LIN {X 0,Y 97.337,Z 845.58,A -85,B 0,C 180,E1 -28950.042,E2 -28950.042} C_VEL
LIN {X 0,Y 109.407,Z 841.998,A -85,B 0,C 180,E1 -28954.063,E2 -28954.063} C_VEL
LIN {X 0,Y 115.747,Z 839.589,A -85,B 0,C 180,E1 -28955.608,E2 -28955.608} C_VEL
LIN {X 0,Y 117.858,Z 838.675,A -85,B 0,C 180,E1 -28956.642,E2 -28956.642} C_VEL
LIN {X 0,Y 108.454,Z 842.054,A -85,B 0,C 180,E1 -28959.119,E2 -28959.119} C_VEL
LIN {X 0,Y 95.133,Z 845.441,A -85,B 0,C 180,E1 -28963.809,E2 -28963.809} C_VEL
LIN {X 0,Y 86.195,Z 846.778,A -85,B 0,C 180,E1 -28968.064,E2 -28968.064} C_VEL
LIN {X 0,Y 76.127,Z 847.276,A -85,B 0,C 180,E1 -28974.702,E2 -28974.702} C_VEL
LIN {X 0,Y 70.276,Z 846.865,A -85,B 0,C 180,E1 -28980.071,E2 -28980.071} C_VEL
LIN {X 0,Y 63.905,Z 845.572,A -85,B 0,C 180,E1 -28988.222,E2 -28988.222} C_VEL
LIN {X 0,Y 57.877,Z 842.432,A -85,B 0,C 180,E1 -29001.363,E2 -29001.363} C_VEL
LIN {X 0,Y 55.288,Z 838.085,A -85,B 0,C 180,E1 -29014.89,E2 -29014.89} C_VEL
LIN {X 0,Y 55.324,Z 833.064,A -85,B 0,C 180,E1 -29026.92,E2 -29026.92} C_VEL
LIN {X 0,Y 56.871,Z 827.685,A -85,B 0,C 180,E1 -29036.869,E2 -29036.869} C_VEL
LIN {X 0,Y 59.908,Z 820.393,A -85,B 0,C 180,E1 -29047.051,E2 -29047.051} C_VEL
LIN {X 0,Y 60.928,Z 818.162,A -85,B 0,C 180,E1 -29049.601,E2 -29049.601} C_VEL
LIN {X 0,Y 62.142,Z 814.385,A -85,B 0,C 180,E1 -29053.604,E2 -29053.604} C_VEL
LIN {X 0,Y 62.854,Z 807.647,A -85,B 0,C 180,E1 -29060.19,E2 -29060.19} C_VEL
LIN {X 0,Y 64.057,Z 800.304,A -85,B 0,C 180,E1 -29066.256,E2 -29066.256} C_VEL
LIN {X 0,Y 65.919,Z 795.617,A -85,B 0,C 180,E1 -29069.117,E2 -29069.117} C_VEL
LIN {X 0,Y 70.749,Z 785.494,A -85,B 0,C 180,E1 -29073.493,E2 -29073.493} C_VEL
LIN {X 0,Y 71.926,Z 778.933,A -85,B 0,C 180,E1 -29076.609,E2 -29076.609} C_VEL
LIN {X 0,Y 70.875,Z 778.62,A -85,B 0,C 180,E1 -29077.433,E2 -29077.433} C_VEL
LIN {X 0,Y 64.084,Z 778.084,A -85,B 0,C 180,E1 -29082.673,E2 -29082.673} C_VEL
LIN {X 0,Y 59.157,Z 776.717,A -85,B 0,C 180,E1 -29088.122,E2 -29088.122} C_VEL
LIN {X 0,Y 54.146,Z 776.16,A -85,B 0,C 180,E1 -29094.693,E2 -29094.693} C_VEL
LIN {X 0,Y 52.689,Z 774.473,A -85,B 0,C 180,E1 -29098.644,E2 -29098.644} C_VEL
LIN {X 0,Y 52.676,Z 779.282,A -85,B 0,C 180,E1 -29111.848,E2 -29111.848} C_VEL
LIN {X 0,Y 55.548,Z 783.057,A -85,B 0,C 180,E1 -29125.331,E2 -29125.331} C_VEL
LIN {X 0,Y 61,Z 785.546,A -85,B 0,C 180,E1 -29137.185,E2 -29137.185} C_VEL
LIN {X 0,Y 65.827,Z 786.444,A -85,B 0,C 180,E1 -29143.932,E2 -29143.932} C_VEL
LIN {X 0,Y 71.43,Z 786.807,A -85,B 0,C 180,E1 -29149.721,E2 -29149.721} C_VEL
LIN {X 0,Y 77.758,Z 786.531,A -85,B 0,C 180,E1 -29154.815,E2 -29154.815} C_VEL
LIN {X 0,Y 86.181,Z 785.381,A -85,B 0,C 180,E1 -29160.001,E2 -29160.001} C_VEL
LIN {X 0,Y 95.086,Z 783.29,A -85,B 0,C 180,E1 -29164.239,E2 -29164.239} C_VEL
LIN {X 0,Y 98.897,Z 782.143,A -85,B 0,C 180,E1 -29165.777,E2 -29165.777} C_VEL
LIN {X 0,Y 102.271,Z 781.127,A -85,B 0,C 180,E1 -29167.9,E2 -29167.9} C_VEL
LIN {X 0,Y 103.122,Z 781.36,A -85,B 0,C 180,E1 -29171.798,E2 -29171.798} C_VEL
LIN {X 0,Y 102.209,Z 782.608,A -85,B 0,C 180,E1 -29175.965,E2 -29175.965} C_VEL
LIN {X 0,Y 100.508,Z 784.208,A -85,B 0,C 180,E1 -29179.374,E2 -29179.374} C_VEL
LIN {X 0,Y 91.817,Z 788.201,A -85,B 0,C 180,E1 -29183.284,E2 -29183.284} C_VEL
LIN {X 0,Y 80.528,Z 792.377,A -85,B 0,C 180,E1 -29189.217,E2 -29189.217} C_VEL
LIN {X 0,Y 70.349,Z 795.196,A -85,B 0,C 180,E1 -29196.94,E2 -29196.94} C_VEL
LIN {X 0,Y 66.904,Z 796.068,A -85,B 0,C 180,E1 -29200.409,E2 -29200.409} C_VEL
LIN {X 0,Y 61.403,Z 806.889,A -85,B 0,C 180,E1 -29206.623,E2 -29206.623} C_VEL
LIN {X 0,Y 56.665,Z 815.69,A -85,B 0,C 180,E1 -29213.901,E2 -29213.901} C_VEL
LIN {X 0,Y 52.334,Z 824.279,A -85,B 0,C 180,E1 -29224.118,E2 -29224.118} C_VEL
LIN {X 0,Y 49.821,Z 831.224,A -85,B 0,C 180,E1 -29235.704,E2 -29235.704} C_VEL
LIN {X 0,Y 49.137,Z 835.892,A -85,B 0,C 180,E1 -29245.895,E2 -29245.895} C_VEL
LIN {X 0,Y 49.267,Z 838.605,A -85,B 0,C 180,E1 -29253.059,E2 -29253.059} C_VEL
LIN {X 0,Y 50.036,Z 842.482,A -85,B 0,C 180,E1 -29266.31,E2 -29266.31} C_VEL
LIN {X 0,Y 54.162,Z 845.868,A -85,B 0,C 180,E1 -29281.263,E2 -29281.263} C_VEL
LIN {X 0,Y 61.486,Z 847.824,A -85,B 0,C 180,E1 -29293.295,E2 -29293.295} C_VEL
LIN {X 0,Y 71.066,Z 848.501,A -85,B 0,C 180,E1 -29302.288,E2 -29302.288} C_VEL
LIN {X 0,Y 82.054,Z 847.895,A -85,B 0,C 180,E1 -29308.921,E2 -29308.921} C_VEL
LIN {X 0,Y 94,Z 845.97,A -85,B 0,C 180,E1 -29313.785,E2 -29313.785} C_VEL
LIN {X 0,Y 100.238,Z 844.484,A -85,B 0,C 180,E1 -29315.704,E2 -29315.704} C_VEL
LIN {X 0,Y 100.894,Z 844.252,A -85,B 0,C 180,E1 -29316.994,E2 -29316.994} C_VEL
LIN {X 0,Y 88.164,Z 846.641,A -85,B 0,C 180,E1 -29321.405,E2 -29321.405} C_VEL
LIN {X 0,Y 79.941,Z 847.375,A -85,B 0,C 180,E1 -29325.242,E2 -29325.242} C_VEL
LIN {X 0,Y 71.204,Z 847.416,A -85,B 0,C 180,E1 -29330.737,E2 -29330.737} C_VEL
LIN {X 0,Y 61.361,Z 846.218,A -85,B 0,C 180,E1 -29339.999,E2 -29339.999} C_VEL
LIN {X 0,Y 54.212,Z 843.827,A -85,B 0,C 180,E1 -29351.212,E2 -29351.212} C_VEL
LIN {X 0,Y 49.577,Z 840.062,A -85,B 0,C 180,E1 -29365.167,E2 -29365.167} C_VEL
LIN {X 0,Y 48.011,Z 835.37,A -85,B 0,C 180,E1 -29379.356,E2 -29379.356} C_VEL
LIN {X 0,Y 49.024,Z 829.528,A -85,B 0,C 180,E1 -29393.16,E2 -29393.16} C_VEL
LIN {X 0,Y 51.417,Z 823.332,A -85,B 0,C 180,E1 -29404.099,E2 -29404.099} C_VEL
LIN {X 0,Y 55.431,Z 815.299,A -85,B 0,C 180,E1 -29414.374,E2 -29414.374} C_VEL
LIN {X 0,Y 60.999,Z 805.035,A -85,B 0,C 180,E1 -29423.388,E2 -29423.388} C_VEL
LIN {X 0,Y 65.919,Z 795.617,A -85,B 0,C 180,E1 -29429.117,E2 -29429.117} C_VEL
LIN {X 0,Y 66.46,Z 793.686,A -85,B 0,C 180,E1 -29430.333,E2 -29430.333} C_VEL
LIN {X 0,Y 65.983,Z 790.673,A -85,B 0,C 180,E1 -29432.816,E2 -29432.816} C_VEL
LIN {X 0,Y 64.886,Z 786.315,A -85,B 0,C 180,E1 -29436.529,E2 -29436.529} C_VEL
LIN {X 0,Y 64.896,Z 785.615,A -85,B 0,C 180,E1 -29436.997,E2 -29436.997} C_VEL
LIN {X 0,Y 64.976,Z 784.515,A -85,B 0,C 180,E1 -29437.69,E2 -29437.69} C_VEL
LIN {X 0,Y 52.577,Z 782.682,A -85,B 0,C 180,E1 -29450.664,E2 -29450.664} C_VEL
LIN {X 0,Y 50.05,Z 781.938,A -85,B 0,C 180,E1 -29454.919,E2 -29454.919} C_VEL
LIN {X 0,Y 48.232,Z 780.916,A -85,B 0,C 180,E1 -29459.042,E2 -29459.042} C_VEL
LIN {X 0,Y 46.361,Z 780.459,A -85,B 0,C 180,E1 -29463.383,E2 -29463.383} C_VEL
LIN {X 0,Y 45.36,Z 778.621,A -85,B 0,C 180,E1 -29468.939,E2 -29468.939} C_VEL
LIN {X 0,Y 47.662,Z 782.726,A -85,B 0,C 180,E1 -29483.857,E2 -29483.857} C_VEL
LIN {X 0,Y 53.163,Z 785.8,A -85,B 0,C 180,E1 -29497.736,E2 -29497.736} C_VEL
LIN {X 0,Y 58.848,Z 787.189,A -85,B 0,C 180,E1 -29506.182,E2 -29506.182} C_VEL
LIN {X 0,Y 66.591,Z 787.888,A -85,B 0,C 180,E1 -29513.943,E2 -29513.943} C_VEL
LIN {X 0,Y 77.331,Z 787.449,A -85,B 0,C 180,E1 -29521.316,E2 -29521.316} C_VEL
LIN {X 0,Y 84.667,Z 786.379,A -85,B 0,C 180,E1 -29525.043,E2 -29525.043} C_VEL
LIN {X 0,Y 93.622,Z 784.354,A -85,B 0,C 180,E1 -29528.635,E2 -29528.635} C_VEL
LIN {X 0,Y 96.122,Z 783.845,A -85,B 0,C 180,E1 -29530.533,E2 -29530.533} C_VEL
LIN {X 0,Y 96.146,Z 784.213,A -85,B 0,C 180,E1 -29532.668,E2 -29532.668} C_VEL
LIN {X 0,Y 95.065,Z 785.304,A -85,B 0,C 180,E1 -29536.033,E2 -29536.033} C_VEL
LIN {X 0,Y 92.068,Z 786.659,A -85,B 0,C 180,E1 -29537.779,E2 -29537.779} C_VEL
LIN {X 0,Y 83.149,Z 789.928,A -85,B 0,C 180,E1 -29541.597,E2 -29541.597} C_VEL
LIN {X 0,Y 71.606,Z 793.148,A -85,B 0,C 180,E1 -29547.947,E2 -29547.947} C_VEL
LIN {X 0,Y 61.147,Z 795.333,A -85,B 0,C 180,E1 -29556.773,E2 -29556.773} C_VEL
LIN {X 0,Y 55.344,Z 805.988,A -85,B 0,C 180,E1 -29563.094,E2 -29563.094} C_VEL
LIN {X 0,Y 50.173,Z 814.923,A -85,B 0,C 180,E1 -29570.919,E2 -29570.919} C_VEL
LIN {X 0,Y 45.436,Z 823.576,A -85,B 0,C 180,E1 -29582.347,E2 -29582.347} C_VEL
LIN {X 0,Y 42.75,Z 830.558,A -85,B 0,C 180,E1 -29595.719,E2 -29595.719} C_VEL
LIN {X 0,Y 42.189,Z 836.105,A -85,B 0,C 180,E1 -29609.995,E2 -29609.995} C_VEL
LIN {X 0,Y 42.383,Z 839.021,A -85,B 0,C 180,E1 -29619.54,E2 -29619.54} C_VEL
LIN {X 0,Y 43.338,Z 841.409,A -85,B 0,C 180,E1 -29628.92,E2 -29628.92} C_VEL
LIN {X 0,Y 48.259,Z 845.009,A -85,B 0,C 180,E1 -29645.623,E2 -29645.623} C_VEL
LIN {X 0,Y 56.537,Z 847.275,A -85,B 0,C 180,E1 -29658.226,E2 -29658.226} C_VEL
LIN {X 0,Y 66.96,Z 848.237,A -85,B 0,C 180,E1 -29667.099,E2 -29667.099} C_VEL
LIN {X 0,Y 79.607,Z 847.804,A -85,B 0,C 180,E1 -29673.805,E2 -29673.805} C_VEL
LIN {X 0,Y 84.784,Z 847.24,A -85,B 0,C 180,E1 -29675.752,E2 -29675.752} C_VEL
LIN {X 0,Y 85.312,Z 847.12,A -85,B 0,C 180,E1 -29677.097,E2 -29677.097} C_VEL
LIN {X 0,Y 72,Z 847.759,A -85,B 0,C 180,E1 -29682.971,E2 -29682.971} C_VEL
LIN {X 0,Y 64.772,Z 847.344,A -85,B 0,C 180,E1 -29687.546,E2 -29687.546} C_VEL
LIN {X 0,Y 56.435,Z 846.07,A -85,B 0,C 180,E1 -29694.992,E2 -29694.992} C_VEL
LIN {X 0,Y 47.475,Z 842.995,A -85,B 0,C 180,E1 -29708.512,E2 -29708.512} C_VEL
LIN {X 0,Y 42.448,Z 838.838,A -85,B 0,C 180,E1 -29724.45,E2 -29724.45} C_VEL
LIN {X 0,Y 40.969,Z 834.012,A -85,B 0,C 180,E1 -29740.189,E2 -29740.189} C_VEL
LIN {X 0,Y 42.328,Z 827.781,A -85,B 0,C 180,E1 -29756.114,E2 -29756.114} C_VEL
LIN {X 0,Y 46.034,Z 819.842,A -85,B 0,C 180,E1 -29770.545,E2 -29770.545} C_VEL
LIN {X 0,Y 50.792,Z 811.433,A -85,B 0,C 180,E1 -29780.859,E2 -29780.859} C_VEL
LIN {X 0,Y 56.667,Z 801.359,A -85,B 0,C 180,E1 -29789.122,E2 -29789.122} C_VEL
LIN {X 0,Y 62.557,Z 790.472,A -85,B 0,C 180,E1 -29795,E2 -29795} C_VEL
LIN {X 0,Y 64.896,Z 785.615,A -85,B 0,C 180,E1 -29796.997,E2 -29796.997} C_VEL
LIN {X 0,Y 64.321,Z 784.532,A -85,B 0,C 180,E1 -29798.144,E2 -29798.144} C_VEL
LIN {X 0,Y 62.594,Z 784.124,A -85,B 0,C 180,E1 -29799.71,E2 -29799.71} C_VEL
LIN {X 0,Y 59.438,Z 784.737,A -85,B 0,C 180,E1 -29801.741,E2 -29801.741} C_VEL
LIN {X 0,Y 51.676,Z 787.896,A -85,B 0,C 180,E1 -29806.496,E2 -29806.496} C_VEL
LIN {X 0,Y 48.765,Z 788.348,A -85,B 0,C 180,E1 -29809.575,E2 -29809.575} C_VEL
LIN {X 0,Y 48.234,Z 788.279,A -85,B 0,C 180,E1 -29810.273,E2 -29810.273} C_VEL
LIN {X 0,Y 46.147,Z 787.8,A -85,B 0,C 180,E1 -29813.971,E2 -29813.971} C_VEL
LIN {X 0,Y 44.339,Z 786.87,A -85,B 0,C 180,E1 -29818.398,E2 -29818.398} C_VEL
LIN {X 0,Y 42.292,Z 786.267,A -85,B 0,C 180,E1 -29823.813,E2 -29823.813} C_VEL
LIN {X 0,Y 39.709,Z 783.567,A -85,B 0,C 180,E1 -29838.969,E2 -29838.969} C_VEL
LIN {X 0,Y 39.996,Z 782.339,A -85,B 0,C 180,E1 -29842.772,E2 -29842.772} C_VEL
LIN {X 0,Y 45.317,Z 785.818,A -85,B 0,C 180,E1 -29858.526,E2 -29858.526} C_VEL
LIN {X 0,Y 50.472,Z 787.442,A -85,B 0,C 180,E1 -29867.104,E2 -29867.104} C_VEL
LIN {X 0,Y 56.536,Z 788.528,A -85,B 0,C 180,E1 -29874.011,E2 -29874.011} C_VEL
LIN {X 0,Y 63.833,Z 789.022,A -85,B 0,C 180,E1 -29880.001,E2 -29880.001} C_VEL
LIN {X 0,Y 73.049,Z 788.763,A -85,B 0,C 180,E1 -29885.522,E2 -29885.522} C_VEL
LIN {X 0,Y 85.904,Z 787.008,A -85,B 0,C 180,E1 -29890.953,E2 -29890.953} C_VEL
LIN {X 0,Y 89.267,Z 786.298,A -85,B 0,C 180,E1 -29892.095,E2 -29892.095} C_VEL
LIN {X 0,Y 88.473,Z 786.839,A -85,B 0,C 180,E1 -29893.788,E2 -29893.788} C_VEL
LIN {X 0,Y 80.76,Z 789.338,A -85,B 0,C 180,E1 -29896.805,E2 -29896.805} C_VEL
LIN {X 0,Y 68.515,Z 792.346,A -85,B 0,C 180,E1 -29902.597,E2 -29902.597} C_VEL
LIN {X 0,Y 57.301,Z 794.094,A -85,B 0,C 180,E1 -29910.84,E2 -29910.84} C_VEL
LIN {X 0,Y 55.843,Z 794.237,A -85,B 0,C 180,E1 -29912.261,E2 -29912.261} C_VEL
LIN {X 0,Y 49.56,Z 804.974,A -85,B 0,C 180,E1 -29918.738,E2 -29918.738} C_VEL
LIN {X 0,Y 43.888,Z 813.982,A -85,B 0,C 180,E1 -29927.105,E2 -29927.105} C_VEL
LIN {X 0,Y 39.349,Z 821.447,A -85,B 0,C 180,E1 -29937.594,E2 -29937.594} C_VEL
LIN {X 0,Y 35.981,Z 828.804,A -85,B 0,C 180,E1 -29952.957,E2 -29952.957} C_VEL
LIN {X 0,Y 35.21,Z 834.649,A -85,B 0,C 180,E1 -29969.994,E2 -29969.994} C_VEL
LIN {X 0,Y 35.528,Z 837.689,A -85,B 0,C 180,E1 -29981.403,E2 -29981.403} C_VEL
LIN {X 0,Y 39.191,Z 842.35,A -85,B 0,C 180,E1 -30002.54,E2 -30002.54} C_VEL
LIN {X 0,Y 47.015,Z 845.54,A -85,B 0,C 180,E1 -30018.36,E2 -30018.36} C_VEL
LIN {X 0,Y 57.584,Z 847.407,A -85,B 0,C 180,E1 -30028.679,E2 -30028.679} C_VEL
LIN {X 0,Y 69.464,Z 848.012,A -85,B 0,C 180,E1 -30035.576,E2 -30035.576} C_VEL
LIN {X 0,Y 71.164,Z 848,A -85,B 0,C 180,E1 -30036.731,E2 -30036.731} C_VEL
LIN {X 0,Y 58.589,Z 847.04,A -85,B 0,C 180,E1 -30043.652,E2 -30043.652} C_VEL
LIN {X 0,Y 49.39,Z 845.219,A -85,B 0,C 180,E1 -30051.818,E2 -30051.818} C_VEL
LIN {X 0,Y 40.483,Z 841.791,A -85,B 0,C 180,E1 -30065.86,E2 -30065.86} C_VEL
LIN {X 0,Y 35.359,Z 837.422,A -85,B 0,C 180,E1 -30083.422,E2 -30083.422} C_VEL
LIN {X 0,Y 33.963,Z 832.35,A -85,B 0,C 180,E1 -30101.915,E2 -30101.915} C_VEL
LIN {X 0,Y 35.339,Z 827.03,A -85,B 0,C 180,E1 -30117.472,E2 -30117.472} C_VEL
LIN {X 0,Y 38.697,Z 820.325,A -85,B 0,C 180,E1 -30131.699,E2 -30131.699} C_VEL
LIN {X 0,Y 43.789,Z 812.017,A -85,B 0,C 180,E1 -30143.526,E2 -30143.526} C_VEL
LIN {X 0,Y 50.233,Z 801.797,A -85,B 0,C 180,E1 -30152.734,E2 -30152.734} C_VEL
LIN {X 0,Y 56.066,Z 791.883,A -85,B 0,C 180,E1 -30158.482,E2 -30158.482} C_VEL
LIN {X 0,Y 56.955,Z 790.27,A -85,B 0,C 180,E1 -30159.196,E2 -30159.196} C_VEL
LIN {X 0,Y 57.024,Z 789.715,A -85,B 0,C 180,E1 -30159.617,E2 -30159.617} C_VEL
LIN {X 0,Y 48.234,Z 788.279,A -85,B 0,C 180,E1 -30170.273,E2 -30170.273} C_VEL
LIN {X 0,Y 45.683,Z 788.282,A -85,B 0,C 180,E1 -30174.062,E2 -30174.062} C_VEL
LIN {X 0,Y 37.471,Z 790.668,A -85,B 0,C 180,E1 -30188.534,E2 -30188.534} C_VEL
LIN {X 0,Y 36.204,Z 790.309,A -85,B 0,C 180,E1 -30194.31,E2 -30194.31} C_VEL
LIN {X 0,Y 35.712,Z 789.101,A -85,B 0,C 180,E1 -30201.932,E2 -30201.932} C_VEL
LIN {X 0,Y 35.858,Z 788.529,A -85,B 0,C 180,E1 -30203.988,E2 -30203.988} C_VEL
LIN {X 0,Y 35.861,Z 787.845,A -85,B 0,C 180,E1 -30210.14,E2 -30210.14} C_VEL
LIN {X 0,Y 36.78,Z 786.234,A -85,B 0,C 180,E1 -30217.534,E2 -30217.534} C_VEL
LIN {X 0,Y 37.479,Z 785.595,A -85,B 0,C 180,E1 -30219.667,E2 -30219.667} C_VEL
LIN {X 0,Y 43.694,Z 787.83,A -85,B 0,C 180,E1 -30230.745,E2 -30230.745} C_VEL
LIN {X 0,Y 52.37,Z 789.488,A -85,B 0,C 180,E1 -30240.001,E2 -30240.001} C_VEL
LIN {X 0,Y 63.816,Z 790.186,A -85,B 0,C 180,E1 -30247.603,E2 -30247.603} C_VEL
LIN {X 0,Y 74.312,Z 789.681,A -85,B 0,C 180,E1 -30252.292,E2 -30252.292} C_VEL
LIN {X 0,Y 72.45,Z 790.283,A -85,B 0,C 180,E1 -30254.047,E2 -30254.047} C_VEL
LIN {X 0,Y 59.89,Z 792.403,A -85,B 0,C 180,E1 -30260.142,E2 -30260.142} C_VEL
LIN {X 0,Y 50.786,Z 793.238,A -85,B 0,C 180,E1 -30267.011,E2 -30267.011} C_VEL
LIN {X 0,Y 44.145,Z 803.885,A -85,B 0,C 180,E1 -30273.291,E2 -30273.291} C_VEL
LIN {X 0,Y 37.858,Z 813.022,A -85,B 0,C 180,E1 -30282.041,E2 -30282.041} C_VEL
LIN {X 0,Y 32.724,Z 820.6,A -85,B 0,C 180,E1 -30293.792,E2 -30293.792} C_VEL
LIN {X 0,Y 28.92,Z 828.043,A -85,B 0,C 180,E1 -30312.308,E2 -30312.308} C_VEL
LIN {X 0,Y 28.202,Z 833.034,A -85,B 0,C 180,E1 -30329.992,E2 -30329.992} C_VEL
LIN {X 0,Y 28.738,Z 836.282,A -85,B 0,C 180,E1 -30344.148,E2 -30344.148} C_VEL
LIN {X 0,Y 33.497,Z 841.221,A -85,B 0,C 180,E1 -30369,E2 -30369} C_VEL
LIN {X 0,Y 42.662,Z 844.671,A -85,B 0,C 180,E1 -30385.445,E2 -30385.445} C_VEL
LIN {X 0,Y 54.241,Z 846.862,A -85,B 0,C 180,E1 -30395.083,E2 -30395.083} C_VEL
LIN {X 0,Y 55.033,Z 846.902,A -85,B 0,C 180,E1 -30397.472,E2 -30397.472} C_VEL
LIN {X 0,Y 43.313,Z 844.314,A -85,B 0,C 180,E1 -30406.775,E2 -30406.775} C_VEL
LIN {X 0,Y 34.552,Z 840.88,A -85,B 0,C 180,E1 -30419.998,E2 -30419.998} C_VEL
LIN {X 0,Y 28.16,Z 835.625,A -85,B 0,C 180,E1 -30442.761,E2 -30442.761} C_VEL
LIN {X 0,Y 27.006,Z 830.633,A -85,B 0,C 180,E1 -30463.821,E2 -30463.821} C_VEL
LIN {X 0,Y 29.173,Z 824.552,A -85,B 0,C 180,E1 -30484.044,E2 -30484.044} C_VEL
LIN {X 0,Y 34.168,Z 816.511,A -85,B 0,C 180,E1 -30501.446,E2 -30501.446} C_VEL
LIN {X 0,Y 40.651,Z 807.233,A -85,B 0,C 180,E1 -30513.151,E2 -30513.151} C_VEL
LIN {X 0,Y 47.83,Z 796.449,A -85,B 0,C 180,E1 -30521.13,E2 -30521.13} C_VEL
LIN {X 0,Y 48.617,Z 795.158,A -85,B 0,C 180,E1 -30521.83,E2 -30521.83} C_VEL
LIN {X 0,Y 38.111,Z 791.992,A -85,B 0,C 180,E1 -30543.595,E2 -30543.595} C_VEL
LIN {X 0,Y 36.204,Z 790.309,A -85,B 0,C 180,E1 -30554.31,E2 -30554.31} C_VEL
LIN {X 0,Y 35.398,Z 789.859,A -85,B 0,C 180,E1 -30560.518,E2 -30560.518} C_VEL
LIN {X 0,Y 33.879,Z 791.155,A -85,B 0,C 180,E1 -30582.724,E2 -30582.724} C_VEL
LIN {X 0,Y 34.916,Z 790.692,A -85,B 0,C 180,E1 -30589.095,E2 -30589.095} C_VEL
LIN {X 0,Y 37.438,Z 788.979,A -85,B 0,C 180,E1 -30595.811,E2 -30595.811} C_VEL
LIN {X 0,Y 38.265,Z 788.338,A -85,B 0,C 180,E1 -30597.139,E2 -30597.139} C_VEL
LIN {X 0,Y 50.495,Z 790.632,A -85,B 0,C 180,E1 -30608.002,E2 -30608.002} C_VEL
LIN {X 0,Y 57.459,Z 791.188,A -85,B 0,C 180,E1 -30611.886,E2 -30611.886} C_VEL
LIN {X 0,Y 57.805,Z 791.406,A -85,B 0,C 180,E1 -30613.419,E2 -30613.419} C_VEL
LIN {X 0,Y 46.246,Z 792.217,A -85,B 0,C 180,E1 -30620.669,E2 -30620.669} C_VEL
LIN {X 0,Y 39.237,Z 802.756,A -85,B 0,C 180,E1 -30626.404,E2 -30626.404} C_VEL
LIN {X 0,Y 32.25,Z 811.983,A -85,B 0,C 180,E1 -30635.183,E2 -30635.183} C_VEL
LIN {X 0,Y 26.319,Z 819.627,A -85,B 0,C 180,E1 -30648.108,E2 -30648.108} C_VEL
LIN {X 0,Y 21.884,Z 827.174,A -85,B 0,C 180,E1 -30671.257,E2 -30671.257} C_VEL
LIN {X 0,Y 21.243,Z 831.349,A -85,B 0,C 180,E1 -30689.99,E2 -30689.99} C_VEL
LIN {X 0,Y 22.085,Z 834.756,A -85,B 0,C 180,E1 -30708.546,E2 -30708.546} C_VEL
LIN {X 0,Y 26.252,Z 838.835,A -85,B 0,C 180,E1 -30732.001,E2 -30732.001} C_VEL
LIN {X 0,Y 33.418,Z 842.056,A -85,B 0,C 180,E1 -30747.258,E2 -30747.258} C_VEL
LIN {X 0,Y 39.1,Z 843.754,A -85,B 0,C 180,E1 -30753.977,E2 -30753.977} C_VEL
LIN {X 0,Y 40.75,Z 844.105,A -85,B 0,C 180,E1 -30757.483,E2 -30757.483} C_VEL
LIN {X 0,Y 28.287,Z 839.42,A -85,B 0,C 180,E1 -30773.55,E2 -30773.55} C_VEL
LIN {X 0,Y 21.295,Z 834.042,A -85,B 0,C 180,E1 -30799.268,E2 -30799.268} C_VEL
LIN {X 0,Y 20.316,Z 827.949,A -85,B 0,C 180,E1 -30831.09,E2 -30831.09} C_VEL
LIN {X 0,Y 23.959,Z 821.187,A -85,B 0,C 180,E1 -30855.854,E2 -30855.854} C_VEL
LIN {X 0,Y 29.788,Z 813.542,A -85,B 0,C 180,E1 -30871.699,E2 -30871.699} C_VEL
LIN {X 0,Y 37.027,Z 804.242,A -85,B 0,C 180,E1 -30882.106,E2 -30882.106} C_VEL
LIN {X 0,Y 39.49,Z 800.902,A -85,B 0,C 180,E1 -30884.619,E2 -30884.619} C_VEL
LIN {X 0,Y 40.257,Z 799.493,A -85,B 0,C 180,E1 -30885.817,E2 -30885.817} C_VEL
LIN {X 0,Y 33.617,Z 797.483,A -85,B 0,C 180,E1 -30903.258,E2 -30903.258} C_VEL
LIN {X 0,Y 32.061,Z 793.373,A -85,B 0,C 180,E1 -30934,E2 -30934} C_VEL
LIN {X 0,Y 33.572,Z 791.626,A -85,B 0,C 180,E1 -30942.932,E2 -30942.932} C_VEL
LIN {X 0,Y 34.916,Z 790.692,A -85,B 0,C 180,E1 -30949.095,E2 -30949.095} C_VEL
LIN {X 0,Y 35.607,Z 790.713,A -85,B 0,C 180,E1 -30953.043,E2 -30953.043} C_VEL
LIN {X 0,Y 35.845,Z 792.068,A -85,B 0,C 180,E1 -30958.201,E2 -30958.201} C_VEL
LIN {X 0,Y 35.341,Z 794.998,A -85,B 0,C 180,E1 -30964.214,E2 -30964.214} C_VEL
LIN {X 0,Y 34.498,Z 797.751,A -85,B 0,C 180,E1 -30968.54,E2 -30968.54} C_VEL
LIN {X 0,Y 32.54,Z 802.596,A -85,B 0,C 180,E1 -30975.26,E2 -30975.26} C_VEL
LIN {X 0,Y 29.918,Z 807.402,A -85,B 0,C 180,E1 -30981.531,E2 -30981.531} C_VEL
LIN {X 0,Y 27.618,Z 810.469,A -85,B 0,C 180,E1 -30985.199,E2 -30985.199} C_VEL
LIN {X 0,Y 20.342,Z 818.639,A -85,B 0,C 180,E1 -30998.965,E2 -30998.965} C_VEL
LIN {X 0,Y 14.842,Z 826.339,A -85,B 0,C 180,E1 -31029.4,E2 -31029.4} C_VEL
LIN {X 0,Y 14.745,Z 831.434,A -85,B 0,C 180,E1 -31063.787,E2 -31063.787} C_VEL
LIN {X 0,Y 19.191,Z 836.118,A -85,B 0,C 180,E1 -31097.074,E2 -31097.074} C_VEL
LIN {X 0,Y 25.52,Z 839.177,A -85,B 0,C 180,E1 -31112.395,E2 -31112.395} C_VEL
LIN {X 0,Y 27.208,Z 839.818,A -85,B 0,C 180,E1 -31116.894,E2 -31116.894} C_VEL
LIN {X 0,Y 16.809,Z 834.285,A -85,B 0,C 180,E1 -31139.996,E2 -31139.996} C_VEL
LIN {X 0,Y 13.08,Z 827.813,A -85,B 0,C 180,E1 -31186.102,E2 -31186.102} C_VEL
LIN {X 0,Y 16.855,Z 821.386,A -85,B 0,C 180,E1 -31221.236,E2 -31221.236} C_VEL
LIN {X 0,Y 23.905,Z 813.472,A -85,B 0,C 180,E1 -31240.597,E2 -31240.597} C_VEL
LIN {X 0,Y 31.711,Z 804.424,A -85,B 0,C 180,E1 -31250.416,E2 -31250.416} C_VEL
LIN {X 0,Y 30.929,Z 803.431,A -85,B 0,C 180,E1 -31254.648,E2 -31254.648} C_VEL
LIN {X 0,Y 27.107,Z 800.734,A -85,B 0,C 180,E1 -31281.071,E2 -31281.071} C_VEL
LIN {X 0,Y 29.196,Z 797.787,A -85,B 0,C 180,E1 -31304.366,E2 -31304.366} C_VEL
LIN {X 0,Y 33.945,Z 795.134,A -85,B 0,C 180,E1 -31320.002,E2 -31320.002} C_VEL
LIN {X 0,Y 35.169,Z 794.405,A -85,B 0,C 180,E1 -31322.201,E2 -31322.201} C_VEL
LIN {X 0,Y 39.851,Z 792.279,A -85,B 0,C 180,E1 -31330.159,E2 -31330.159} C_VEL
LIN {X 0,Y 41.511,Z 791.288,A -85,B 0,C 180,E1 -31331.923,E2 -31331.923} C_VEL
LIN {X 0,Y 41.12,Z 792.976,A -85,B 0,C 180,E1 -31333.824,E2 -31333.824} C_VEL
LIN {X 0,Y 33.462,Z 803.442,A -85,B 0,C 180,E1 -31339.05,E2 -31339.05} C_VEL
LIN {X 0,Y 27.618,Z 810.469,A -85,B 0,C 180,E1 -31345.199,E2 -31345.199} C_VEL
LIN {X 0,Y 23.665,Z 814.419,A -85,B 0,C 180,E1 -31349.473,E2 -31349.473} C_VEL
LIN {X 0,Y 16.023,Z 820.085,A -85,B 0,C 180,E1 -31357.619,E2 -31357.619} C_VEL
LIN {X 0,Y 10.042,Z 824.13,A -85,B 0,C 180,E1 -31373.337,E2 -31373.337} C_VEL
LIN {X 0,Y 7.423,Z 827.085,A -85,B 0,C 180,E1 -31403.473,E2 -31403.473} C_VEL
LIN {X 0,Y 7.415,Z 828.078,A -85,B 0,C 180,E1 -31416.843,E2 -31416.843} C_VEL
LIN {X 0,Y 10.689,Z 831.87,A -85,B 0,C 180,E1 -31458.883,E2 -31458.883} C_VEL
LIN {X 0,Y 13.184,Z 833.434,A -85,B 0,C 180,E1 -31476.428,E2 -31476.428} C_VEL
LIN {X 0,Y 6.082,Z 827.094,A -85,B 0,C 180,E1 -31537.951,E2 -31537.951} C_VEL
LIN {X 0,Y 11.545,Z 820.118,A -85,B 0,C 180,E1 -31599.987,E2 -31599.987} C_VEL
LIN {X 0,Y 19.427,Z 812.788,A -85,B 0,C 180,E1 -31615.167,E2 -31615.167} C_VEL
LIN {X 0,Y 24.273,Z 807.826,A -85,B 0,C 180,E1 -31619.707,E2 -31619.707} C_VEL
LIN {X 0,Y 23.841,Z 804.097,A -85,B 0,C 180,E1 -31662.858,E2 -31662.858} C_VEL
LIN {X 0,Y 31.176,Z 800.57,A -85,B 0,C 180,E1 -31686.48,E2 -31686.48} C_VEL
LIN {X 0,Y 30.163,Z 802.16,A -85,B 0,C 180,E1 -31687.957,E2 -31687.957} C_VEL
LIN {X 0,Y 21.727,Z 811.347,A -85,B 0,C 180,E1 -31693.936,E2 -31693.936} C_VEL
LIN {X 0,Y 12.323,Z 820.319,A -85,B 0,C 180,E1 -31711.155,E2 -31711.155} C_VEL
LIN {X 0,Y 7.334,Z 827.566,A -85,B 0,C 180,E1 -31769.971,E2 -31769.971} C_VEL
LIN {X 0,Y 7.415,Z 828.078,A -85,B 0,C 180,E1 -31776.843,E2 -31776.843} C_VEL
LIN {X 0,Y 6.495,Z 827.846,A -85,B 0,C 180,E1 -31778.167,E2 -31778.167} C_VEL
LIN {X 0,Y 4.202,Z 825.693,A -85,B 0,C 180,E1 -31750.263,E2 -31750.263} C_VEL
LIN {X 0,Y 9.336,Z 818.998,A -85,B 0,C 180,E1 -31680.811,E2 -31680.811} C_VEL
LIN {X 0,Y 13.842,Z 815.074,A -85,B 0,C 180,E1 -31676.197,E2 -31676.197} C_VEL
LIN {X 0,Y 19.392,Z 810.05,A -85,B 0,C 180,E1 -31675.508,E2 -31675.508} C_VEL
LIN {X 0,Y 20.163,Z 808.92,A -85,B 0,C 180,E1 -31672.495,E2 -31672.495} C_VEL
LIN {X 0,Y 17.36,Z 811.019,A -85,B 0,C 180,E1 -31644.085,E2 -31644.085} C_VEL
LIN {X 0,Y 17.081,Z 811.811,A -85,B 0,C 180,E1 -31636.075,E2 -31636.075} C_VEL
LIN {X 0,Y 7.335,Z 820.045,A -85,B 0,C 180,E1 -31637.656,E2 -31637.656} C_VEL
LIN {X 0,Y 1.093,Z 824.668,A -85,B 0,C 180,E1 -31680.056,E2 -31680.056} C_VEL
LIN {X 0,Y 5.049,Z 822.019,A -85,B 0,C 180,E1 -31680.012,E2 -31680.012} C_VEL
LIN {X 0,Y 13.842,Z 815.074,A -85,B 0,C 180,E1 -31676.197,E2 -31676.197} C_VEL
LIN {X 0,Y 13.842,Z 815.074,A -85,B 0,C 180,E1 -31676.197,E2 -31676.197}

QRS_NEXT_CUT()

QRS_NEXT()
QRS_HOME()

END
